ABB RobotStudio station: ASST2.rsstn

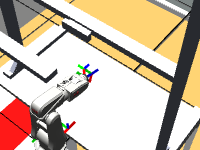
Station ASST2 (saved by RobotStudio format 3)
Controller MTRN4230
  mechanical unit ROB_1: IRB120_3_58__01, 6 joints, base frame (0, 0, 0) mm
Layout (positions relative to the parent item):
  - IRB120_3_58__01 [mechanism, from Robots\IRB120_3_58_G_01.rslib] at (0, 0, 0) mm; joint values [0, 0.0221, 0.2339, 0, 0.0501, 0] (rad or m)
  - assembywohoo [part] at (3015, 1895, -1953) mm, rotated rx 90 ry 0 rz -90 deg
  - Group_1 [graphiccomponentgroup]
    - Group_2 [graphiccomponentgroup]
  - TableCam [frame] at (375, -23, 992) mm
  - ConveyorCam [frame] at (0, 398, 952) mm
Targets, tools, work objects and paths stored in the station, written as RAPID:
! task T_ROB1
MODULE MTRN_Rob_Data
  PERS tooldata tSCup:=[TRUE,[[0,0,65],[1,0,0,0]],[0.5,[0,0,20],[1,0,0,0],0,0,0]];
  PERS wobjdata wTable:=[FALSE,TRUE,"",[[175,0,147],[1,0,0,0]],[[0,0,0],[1,0,0,0]]];
  PERS wobjdata wConv:=[FALSE,TRUE,"",[[50,184,22],[0.5,-0.5,0.5,0.5]],[[1,1,1],[1,0,0,0]]];
  CONST robtarget pTableHome:=[[175,0,147],[0,0,-1,0],[0,0,0,0],[9E9,9E9,9E9,9E9,9E9,9E9]];
  CONST jointtarget jtCalibPos:=[[0,0,0,0,0,0],[9E9,9E9,9E9,9E9,9E9,9E9]];
ENDMODULE

! task T_ROB1
MODULE MTRN4230_Move_Sample
  PROC MoveJSample()
    MoveJ pTableHome,v100,fine,tSCup;
  ENDPROC
  PROC MoveLSample()
    MoveL Offs(pTableHome, 0, 0, 100),v100,fine,tSCup;
  ENDPROC
  PROC MainMove()
    MoveJSample;
    MoveLSample;
  ENDPROC
ENDMODULE

! task T_ROB1
MODULE MTRN_Rob_Proc
  PROC MoveToCalibPos()
    MoveAbsJ jtCalibPos,v400,fine,tool0;
  ENDPROC
ENDMODULE

